// TIA Portal V20 export
FUNCTION_BLOCK "Simulation"   // FB189, LAD
// stored: MemoryReserve 100, Namespace Unit1.Em1, SetENOAutomatically false
   VAR_INPUT
      simulation { ExternalAccessible := 'False'; ExternalVisible := 'False'; ExternalWritable := 'False'} : Bool;
   END_VAR
   VAR
      instActuator { ExternalAccessible := 'False'; ExternalVisible := 'False'; ExternalWritable := 'False'} : Array[0..9] of "Simulation_Actuator";
   END_VAR
BEGIN

REGION Network 1: Two Way Actuator
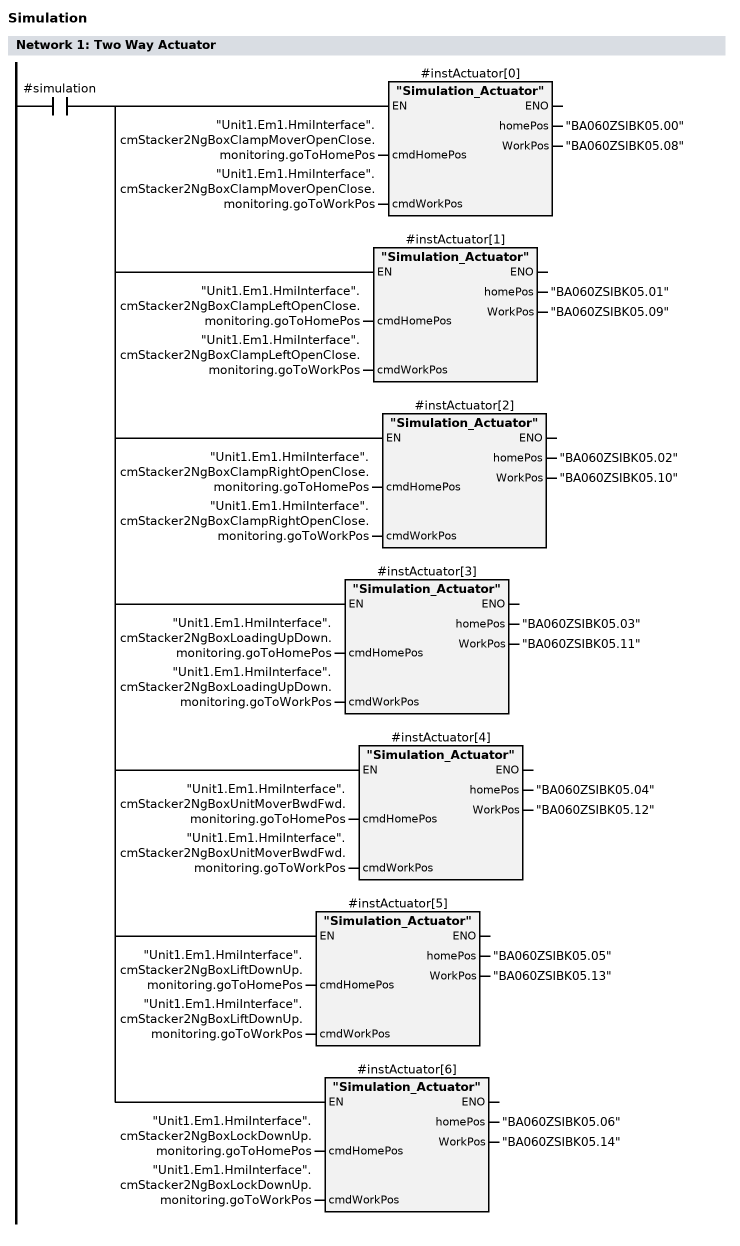
   RUNG wire#powerrail
      Contact( #simulation )
      wire#w1
      #instActuator[0](cmdHomePos := "Unit1.Em1.HmiInterface".cmStacker2NgBoxClampMoverOpenClose.monitoring.goToHomePos, cmdWorkPos := "Unit1.Em1.HmiInterface".cmStacker2NgBoxClampMoverOpenClose.monitoring.goToWorkPos, homePos => "BA060ZSIBK05.00", WorkPos => "BA060ZSIBK05.08")
   END_RUNG
   RUNG wire#w1
      #instActuator[1](cmdHomePos := "Unit1.Em1.HmiInterface".cmStacker2NgBoxClampLeftOpenClose.monitoring.goToHomePos, cmdWorkPos := "Unit1.Em1.HmiInterface".cmStacker2NgBoxClampLeftOpenClose.monitoring.goToWorkPos, homePos => "BA060ZSIBK05.01", WorkPos => "BA060ZSIBK05.09")
   END_RUNG
   RUNG wire#w1
      #instActuator[2](cmdHomePos := "Unit1.Em1.HmiInterface".cmStacker2NgBoxClampRightOpenClose.monitoring.goToHomePos, cmdWorkPos := "Unit1.Em1.HmiInterface".cmStacker2NgBoxClampRightOpenClose.monitoring.goToWorkPos, homePos => "BA060ZSIBK05.02", WorkPos => "BA060ZSIBK05.10")
   END_RUNG
   RUNG wire#w1
      #instActuator[3](cmdHomePos := "Unit1.Em1.HmiInterface".cmStacker2NgBoxLoadingUpDown.monitoring.goToHomePos, cmdWorkPos := "Unit1.Em1.HmiInterface".cmStacker2NgBoxLoadingUpDown.monitoring.goToWorkPos, homePos => "BA060ZSIBK05.03", WorkPos => "BA060ZSIBK05.11")
   END_RUNG
   RUNG wire#w1
      #instActuator[4](cmdHomePos := "Unit1.Em1.HmiInterface".cmStacker2NgBoxUnitMoverBwdFwd.monitoring.goToHomePos, cmdWorkPos := "Unit1.Em1.HmiInterface".cmStacker2NgBoxUnitMoverBwdFwd.monitoring.goToWorkPos, homePos => "BA060ZSIBK05.04", WorkPos => "BA060ZSIBK05.12")
   END_RUNG
   RUNG wire#w1
      #instActuator[5](cmdHomePos := "Unit1.Em1.HmiInterface".cmStacker2NgBoxLiftDownUp.monitoring.goToHomePos, cmdWorkPos := "Unit1.Em1.HmiInterface".cmStacker2NgBoxLiftDownUp.monitoring.goToWorkPos, homePos => "BA060ZSIBK05.05", WorkPos => "BA060ZSIBK05.13")
   END_RUNG
   RUNG wire#w1
      #instActuator[6](cmdHomePos := "Unit1.Em1.HmiInterface".cmStacker2NgBoxLockDownUp.monitoring.goToHomePos, cmdWorkPos := "Unit1.Em1.HmiInterface".cmStacker2NgBoxLockDownUp.monitoring.goToWorkPos, homePos => "BA060ZSIBK05.06", WorkPos => "BA060ZSIBK05.14")
   END_RUNG
   // the same network as SCL:
   IF #simulation THEN
       #instActuator[0](cmdHomePos := "Unit1.Em1.HmiInterface".cmStacker2NgBoxClampMoverOpenClose.monitoring.goToHomePos,   // "Simulation_Actuator"
                        cmdWorkPos := "Unit1.Em1.HmiInterface".cmStacker2NgBoxClampMoverOpenClose.monitoring.goToWorkPos,
                        homePos => "BA060ZSIBK05.00",
                        WorkPos => "BA060ZSIBK05.08");
       #instActuator[1](cmdHomePos := "Unit1.Em1.HmiInterface".cmStacker2NgBoxClampLeftOpenClose.monitoring.goToHomePos,   // "Simulation_Actuator"
                        cmdWorkPos := "Unit1.Em1.HmiInterface".cmStacker2NgBoxClampLeftOpenClose.monitoring.goToWorkPos,
                        homePos => "BA060ZSIBK05.01",
                        WorkPos => "BA060ZSIBK05.09");
       #instActuator[2](cmdHomePos := "Unit1.Em1.HmiInterface".cmStacker2NgBoxClampRightOpenClose.monitoring.goToHomePos,   // "Simulation_Actuator"
                        cmdWorkPos := "Unit1.Em1.HmiInterface".cmStacker2NgBoxClampRightOpenClose.monitoring.goToWorkPos,
                        homePos => "BA060ZSIBK05.02",
                        WorkPos => "BA060ZSIBK05.10");
       #instActuator[3](cmdHomePos := "Unit1.Em1.HmiInterface".cmStacker2NgBoxLoadingUpDown.monitoring.goToHomePos,   // "Simulation_Actuator"
                        cmdWorkPos := "Unit1.Em1.HmiInterface".cmStacker2NgBoxLoadingUpDown.monitoring.goToWorkPos,
                        homePos => "BA060ZSIBK05.03",
                        WorkPos => "BA060ZSIBK05.11");
       #instActuator[4](cmdHomePos := "Unit1.Em1.HmiInterface".cmStacker2NgBoxUnitMoverBwdFwd.monitoring.goToHomePos,   // "Simulation_Actuator"
                        cmdWorkPos := "Unit1.Em1.HmiInterface".cmStacker2NgBoxUnitMoverBwdFwd.monitoring.goToWorkPos,
                        homePos => "BA060ZSIBK05.04",
                        WorkPos => "BA060ZSIBK05.12");
       #instActuator[5](cmdHomePos := "Unit1.Em1.HmiInterface".cmStacker2NgBoxLiftDownUp.monitoring.goToHomePos,   // "Simulation_Actuator"
                        cmdWorkPos := "Unit1.Em1.HmiInterface".cmStacker2NgBoxLiftDownUp.monitoring.goToWorkPos,
                        homePos => "BA060ZSIBK05.05",
                        WorkPos => "BA060ZSIBK05.13");
       #instActuator[6](cmdHomePos := "Unit1.Em1.HmiInterface".cmStacker2NgBoxLockDownUp.monitoring.goToHomePos,   // "Simulation_Actuator"
                        cmdWorkPos := "Unit1.Em1.HmiInterface".cmStacker2NgBoxLockDownUp.monitoring.goToWorkPos,
                        homePos => "BA060ZSIBK05.06",
                        WorkPos => "BA060ZSIBK05.14");
   END_IF;
END_REGION

REGION Network 2 (SCL): Initializing
   IF #simulation AND "JB_Temp".Test_Homing[1] THEN
       "Unit1.Em1.HmiInterface".cmStacker2NgBoxLockDownUp.commands.commandWorkPos := true;

       "JB_Temp".Test_Homing[1] := false;
   END_IF;
END_REGION
END_FUNCTION_BLOCK
